# EPICS autosave request: laudaRE2xx/lIntegralT_settings.req
$(P):DISABLE
$(P):RRATE
$(P):RTEMP
$(P):SET_TEMP
